// TwinCAT 3 PLC project Step0
// ProgramVersion: 3.1.4023.0
// libraries:
//   Tc2_Standard, * (Beckhoff Automation GmbH)
//   Tc2_System, * (Beckhoff Automation GmbH)
//   Tc3_Module, * (Beckhoff Automation GmbH)
// project tree:
//   / PlcTask.TcTTO
//   POUs/ MAIN.TcPOU
//   Task1/ E_SensorBrands.TcDUT, G_VarTask1.TcGVL, P_Task1.TcPOU
//   Task2/ G_VarTask2.TcGVL, Deg2Rad.TcPOU, P_Task2.TcPOU, ST_Timer.TcDUT
//   Task3/ F_UpdateFunc.TcPOU, F_UpdateFunc_REF.TcPOU, G_MotorParameters.TcGVL, P_TASK3.TcPOU, ST_MotorParams.TcDUT
// real-time tasks:
//   TASK PlcTask: cycle T#10ms, priority 20, ADS port 350

CONFIGURATION Step0
    RESOURCE PLC ON TwinCAT3
        TASK PlcTask(INTERVAL := T#10ms, PRIORITY := 20);
        PROGRAM MAIN WITH PlcTask : MAIN;
    END_RESOURCE
END_CONFIGURATION

// ---- Task1/E_SensorBrands.TcDUT
{attribute 'qualified_only'}
{attribute 'strict'}
TYPE E_SensorBrands :
(
	Sick,
	Pilz,
	Parker,
	Bosch 
);
END_TYPE

// ---- Task2/ST_Timer.TcDUT
TYPE ST_Timer :
STRUCT
	bTimerStart : BOOL; 
	tTimerStatus : TIME; 
	bTimerEnd : BOOL; 
	tTimer : TIME := T#10S; 
END_STRUCT
END_TYPE

// ---- Task3/ST_MotorParams.TcDUT
TYPE ST_MotorParams : 
STRUCT
	fMaxSpeed : REAL; 
	fMinSpeed : REAL; 
END_STRUCT
END_TYPE

// ---- Task1/G_VarTask1.TcGVL
{attribute 'qualified_only'}
VAR_GLOBAL
	
tdCurrentDate : DATE_AND_TIME := DT#2023-02-07-13:29:20;
tMyTimer : TIME := T#5S; 
aMyDateArray : ARRAY[1..4] OF DATE := [D#2023-02-07, D#2023-02-08, D#2023-02-09, D#2023-02-10]; 
eSensorOne : E_SensorBrands; 
bTimerStart : BOOL; 
tTimerStatus : TIME; 
bTimerEnd : BOOL; 
tTimer : TIME := T#10S; 
END_VAR

// ---- Task2/G_VarTask2.TcGVL
{attribute 'qualified_only'}
VAR_GLOBAL
	stTimer2 : ST_Timer :=(tTimer:=T#5S); 
	fAngPosDeg : REAL := 90; 
	fAngPosRad : REAL; 
	fPiVal : REAL := 3.14159; 
END_VAR

// ---- Task3/G_MotorParameters.TcGVL
{attribute 'qualified_only'}
VAR_GLOBAL
	stMotorParameters : ST_MotorParams;
	stMotorParameters1 : ST_MotorParams; 
END_VAR

// ---- POUs/MAIN.TcPOU
PROGRAM MAIN
VAR
	pToDate : POINTER TO DATE_AND_TIME; 
	nRefToTime : REFERENCE TO TIME; 
	fbTon : TON := (PT:=G_VarTask1.tTimer);   
	fbTof : TOF := (PT:=G_VarTask2.stTimer2.tTimer); 
	
	bSpeedUpdate : BOOL; 
	fGiveValue : REAL; 
	fbRTrig : R_TRIG;
	bInitiate : BOOL; 
END_VAR

pToDate := ADR(G_VarTask1.tdCurrentDate); 

pToDate^:= DT#2023-02-08-16:23:23; 

nRefToTime REF= G_VarTask1.tMyTimer; 
nRefToTime := T#6S; 


G_VarTask1.aMyDateArray[3] := D#2023-02-25; 
G_VarTask1.eSensorOne := E_SensorBrands.Bosch; 

// TON timer
fbTon(IN:=G_VarTask1.bTimerStart); 
G_VarTask1.bTimerEnd := fbTon.Q; 
G_VarTask1.tTimerStatus := fbTon.ET; 

// TOF timer
fbTof(IN:=G_VarTask2.stTimer2.bTimerStart); 
G_VarTask2.stTimer2.tTimerStatus := fbTof.ET; 
G_VarTask2.stTimer2.bTimerEnd := fbTof.Q; 

G_VarTask2.fAngPosRad := Deg2Rad(fDegIn:=G_VarTask2.fAngPosDeg); 

// Task 3
fbRTrig(CLK := bSpeedUpdate); 
bInitiate := fbRTrig.Q; 

IF bInitiate THEN
	F_UpdateFunc(bUpdateValue:=bSpeedUpdate, fNewValue:=fGiveValue, stMotorParameter := G_MotorParameters.stMotorParameters);
	F_UpdateFunc_REF(bUpdateValue:=bSpeedUpdate, fNewValue:=fGiveValue, stMotorParameter := G_MotorParameters.stMotorParameters1); 
END_IF

// FOR CASE instruction -> article number to sort stuff in to categories

END_PROGRAM

// ---- Task2/Deg2Rad.TcPOU
FUNCTION Deg2Rad : REAL
VAR_INPUT
	fDegIn : REAL; 
END_VAR
VAR
	fRadOut : REAL; 
END_VAR

Deg2Rad := fDegIn * (G_VarTask2.fPiVal/180);

END_FUNCTION

// ---- Task3/F_UpdateFunc.TcPOU
FUNCTION F_UpdateFunc : REAL
VAR_INPUT
	bUpdateValue : BOOL;
	fNewValue : REAL; 
	stMotorParameter : ST_MotorParams; 
END_VAR
VAR
END_VAR

IF bUpdateValue THEN
	stMotorParameter.fMaxSpeed := fNewValue; 
	ELSE
		stMotorParameter.fMaxSpeed := stMotorParameter.fMaxSpeed; 

END_IF;

END_FUNCTION

// ---- Task3/F_UpdateFunc_REF.TcPOU
FUNCTION F_UpdateFunc_REF : REAL
VAR_INPUT
	bUpdateValue : BOOL;
	fNewValue : REAL; 
	stMotorParameter : REFERENCE TO ST_MotorParams; 
END_VAR
VAR
END_VAR

IF bUpdateValue THEN
	stMotorParameter.fMaxSpeed := fNewValue; 
	ELSE
		stMotorParameter.fMaxSpeed := stMotorParameter.fMaxSpeed; 

END_IF;

END_FUNCTION

// ---- Task1/P_Task1.TcPOU
PROGRAM P_Task1
VAR
	pToDate : POINTER TO DATE_AND_TIME; 
END_VAR

pToDate := ADR(G_VarTask1.tdCurrentDate); 

pToDate^:= DT#2023-02-08-15:35:20;

END_PROGRAM

// ---- Task2/P_Task2.TcPOU
PROGRAM P_Task2
VAR
END_VAR

END_PROGRAM

// ---- Task3/P_TASK3.TcPOU
PROGRAM P_TASK3
VAR
	bSpeedUpdate : BOOL; 
	fGiveValue : REAL; 
	fbRTrig : R_TRIG;
	
END_VAR


fbRTrig(CLK := bSpeedUpdate); 
fbRTrig.Q := bSpeedUpdate; 

IF bSpeedUpdate THEN
	F_UpdateFunc(bUpdateValue:=bSpeedUpdate, fNewValue:=fGiveValue, stMotorParameter := G_MotorParameters.stMotorParameters);
	F_UpdateFunc_REF(bUpdateValue:=bSpeedUpdate, fNewValue:=fGiveValue, stMotorParameter := G_MotorParameters.stMotorParameters1); 
END_IF

END_PROGRAM
